// TIA Portal project "ACC_CONVEYOR" (V15)

(* hardware
DEVICE "ACC_CONVEYOR"  TP700 Comfort
   slot 0: "ACC_CONVEYOR"  TP700 Comfort  6AV2 124-0GC01-0AX0  14.0.0.0
   slot 1: "HMI_RT_1"  TP700 Comfort  6AV2 124-0GC01-0AX0  14.0.0.0
   slot 5: "ACC_CONVEYOR.IE_CP_1"  PROFINET Interface  14.0.0.0
      slot 1: "PROFINET Interface_1"  PROFINET Interface
         slot 1: "Port_1"  Port
         slot 2: "Port_2"  Port
   slot 7: "ACC_CONVEYOR.MPI/DP_CP_1"  MPI/DP Interface  14.0.0.0
*)

(* ===== HMI "HMI_RT_1" =====
system functions are stored by id; their names below are inferred from use
connection "SPS_1": IF1 B, SIMATIC S7 300/400 MPI

HMI tags "Default tag table"
   "bottleTypeNow" : Int AT %DB70.DBW10, 1 s
   "handmode_Key" : Byte AT %DB70.DBB38, 1 s
   "handMotorstat" : Int AT %DB70.DBW80, 1 s
   "keyGrup_a" : Byte AT %DB70.DBB0, 1 s
   "bottleTypeSelection" : Int AT %DB70.DBW170, 1 s
   "bottleAccSelect" : Bool AT %DB70.DBX2.5, 1 s
   "activeStart" : Bool AT %M10.0, 1 s
   "lubriState" : Bool AT %M48.0, 1 s
   "lubriCycle" : Int AT %DB51.DBW0, 1 s
   "lubriCycleinSec" : Int AT %DB51.DBW2, 1 s
   "lubriClockOP" : Bool AT %DB70.DBX8.0, 1 s
   "Contrass" : Int, internal

HMI tags "hardware_par"
   "select_motor" : Int AT %DB70.DBW40, 1 s
   "action" : Byte AT %DB70.DBB50, 1 s
   "copy" : Bool AT %DB70.DBX54.0, 1 s
   "towardsMotor" : Int AT %DB70.DBW52, 1 s
   "changeValue" : Int AT %DB70.DBW56, 1 s
   "value" : Real AT %DB70.DBD46, 1 s
   "parameter" : Int AT %DB70.DBW42, 1 s

HMI tags "software_par"
   "param_select" : Int AT %DB70.DBW30, 1 s
   "plc_Input" : Int AT %DB0.DBW30, 1 s
   "plc_Calc" : Int AT %DB0.DBW32, 1 s
   "plc_+fact" : Int AT %DB0.DBW34, 1 s
   "minim_Speed" : Int AT %DB0.DBW20, 1 s
   "maxim_Speed" : Int AT %DB0.DBW22, 1 s
   "corrLL" : Int AT %DB0.DBW8, 1 s
   "corrL" : Int AT %DB0.DBW10, 1 s
   "corrH" : Int AT %DB0.DBW12, 1 s
   "corrHH" : Int AT %DB0.DBW14, 1 s
   "frequency" : Int AT %DB0.DBW40, 1 s
   "rampUpSoft" : Int AT %DB0.DBW16, 1 s
   "rampDownSoft" : Int AT %DB0.DBW18, 1 s
   "fillUpLow" : Int AT %DB0.DBW0, 1 s
   "fillUpNomi" : Int AT %DB0.DBW2, 1 s
   "fillUpHigh" : Int AT %DB0.DBW4, 1 s
   "fillUpMaxi" : Int AT %DB0.DBW6, 1 s
   "statusDataWords" : Int AT %DB0.DBW0, 1 s
   "dbNumber" : Int AT %DB70.DBW180, 1 s
   "dwNumber" : Int AT %DB70.DBW182, 1 s
   "reff_Speed" : Int AT %DB0.DBW28, 1 s

HMI tags "regulation_EBI"
   "speedFiller" : Int AT %DB70.DBW90, 1 s
   "speedEBI" : Int AT %DB70.DBW92, 1 s
   "limOverNomin" : Int AT %DB0.DBW232, 1 s
   "limUnderNomin" : Int AT %DB0.DBW234, 1 s
   "correctionFact" : Int AT %DB0.DBW226, 1 s
   "maxSpeedEBI" : Int AT %DB0.DBW224, 1 s
   "minSpeedEBI" : Int AT %DB0.DBW230, 1 s
   "baseSpeed" : Int AT %DB0.DBW238, 1 s
   "btn_speedchange" : Byte AT %MB143, 1 s

HMI tags "inliner"
   "keyInlinerMode" : Byte AT %DB0.DBB278, 1 s
   "speedfilleer" : Int AT %DB0.DBW272, 1 s
   "speedInliner" : Int AT %DB0.DBW274, 1 s
   "limPosCorr" : Int AT %DB0.DBW246, 1 s
   "limNegCorr" : Int AT %DB0.DBW244, 1 s
   "stepPosCorr" : Int AT %DB0.DBW250, 1 s
   "stepNegCorr" : Int AT %DB0.DBW248, 1 s
   "missBotleRef" : Int AT %DB0.DBW240, 1 s
   "missBottleAct" : Int AT %DB0.DBW242, 1 s
   "actinlinerCorr" : Int AT %DB0.DBW266, 1 s
   "factFeeding" : Int AT %DB0.DBW10, 1 s
   "factInlliner" : Int AT %DB0.DBW12, 1 s
   "factOutfeed" : Int AT %DB0.DBW14, 1 s
   "fillUpFast" : Int AT %DB0.DBW254, 1 s
   "fillUpSlow" : Int AT %DB0.DBW252, 1 s
   "syncCorrStep" : Int AT %DB0.DBW280, 1 s
   "syncAfterBot" : Int AT %DB0.DBW282, 1 s
   "syncCounter" : Int AT %DB0.DBW284, 1 s
   "syncActCorr" : Int AT %DB0.DBW286, 1 s
   "syncStepNr" : Int AT %DB0.DBW288, 1 s

HMI tags "statistic"
   "totalMeasureTime" : DInt AT %DB70.DBD210, 1 s
   "lackBottlesInfeedFiller" : DInt AT %DB70.DBD214, 1 s
   "fillerStop" : DInt AT %DB70.DBD218, 1 s
   "fillerRunningBottleStopClosed" : DInt AT %DB70.DBD222, 1 s
   "startCounting" : Bool AT %DB70.DBX209.2, 1 s
   "stopCounting" : Bool AT %DB70.DBX209.3, 1 s
   "totalBottlesIntoFiller" : DInt AT %DB70.DBD226, 1 s
   "resetCounter" : Bool AT %DB70.DBX209.0, 1 s
   "confirm" : Bool AT %DB70.DBX209.1, 1 s
   "resetCounterState" : Bool AT %DB70.DBX208.0, 1 s

HMI tags "alarm"
   "alarm_1" : Int AT %DB70.DBW126, 1 s
   "alarm_2" : Int AT %DB70.DBW128, 1 s
   "alarm_3" : Int AT %DB70.DBW130, 1 s

HMI tags "monitor"
   "state_mot101" : Int AT %DB1.DBW56, 1 s
   "state_mot102" : Int AT %DB2.DBW56, 1 s
   "state_mot103" : Int AT %DB3.DBW56, 1 s
   "state_mot104" : Int AT %DB4.DBW56, 1 s
   "state_mot105" : Int AT %DB5.DBW56, 1 s
   "state_mot106" : Int AT %DB6.DBW56, 1 s
   "state_mot107" : Int AT %DB7.DBW56, 1 s
   "state_mot108" : Int AT %DB8.DBW56, 1 s
   "state_mot109" : Int AT %DB9.DBW56, 1 s
   "emc_1" : Bool AT %DB70.DBX168.0, 1 s
   "emc_2" : Bool AT %DB70.DBX168.1, 1 s
   "emc_3" : Bool AT %DB70.DBX168.2, 1 s
   "emc_4" : Bool AT %DB70.DBX168.3, 1 s
   "ebi_state" : Int AT %DB70.DBW200, 1 s
   "filler_state" : Int AT %DB70.DBW202, 1 s

discrete alarms
   2: 'MANUAL CONTROL ACTIVATED', class Status, trigger "alarm_1" bit 1
   3: 'LINE RUNNING', class Status, trigger "alarm_1" bit 2
   4: 'INLINER RECEPTABLE FULL', class Warnings, trigger "alarm_1" bit 3
   5: 'EMERGENCY STOP AT PANEL', class Errors, trigger "alarm_1" bit 4
      on Coming: ActivateScreen("121_DISPLAY_STATUS", 0)
   6: 'EMERGENCY STOP AT OUTFEED EBI', class Errors, trigger "alarm_1" bit 5
      on Coming: ActivateScreen("121_DISPLAY_STATUS", 0)
   7: 'EMERGENCY STOP AT INFEED FILLER', class Errors, trigger "alarm_1" bit 6
      on Coming: ActivateScreen("121_DISPLAY_STATUS", 0)
   8: 'FAULT ON MOTOR', class Errors, trigger "alarm_1" bit 7
      on Coming: ActivateScreen("121_DISPLAY_STATUS", 0)
   11: 'ACCUMULATION OUTFEED EBI', class Status, trigger "alarm_1" bit 10
   12: 'EBI NOT READY TO RUN', class Errors, trigger "alarm_1" bit 11
   13: 'EBI BOTTLESTOP MANUALLY OPENED', class Status, trigger "alarm_1" bit 12
   14: 'EBI AT MAXIMUM SPEED', class Warnings, trigger "alarm_1" bit 13
   15: 'EBI AT SYNCHRONISED SPEED', class Status, trigger "alarm_1" bit 14
   16: 'EBI AT MINIMUM SPEED', class Warnings, trigger "alarm_1" bit 15
   21: 'ACCUMULATION OUTFEED FILLER', class Status, trigger "alarm_2" bit 4
   22: 'FILLER STOP', class Errors, trigger "alarm_2" bit 5
   23: 'WAIT FOR FILLER TO OPEN BOTTLESTOP', class Status, trigger "alarm_2" bit 6
   31: 'INLINER RECEPTABLE ALMOT FULL', class Warnings, trigger "alarm_2" bit 14
   32: 'INLINER STOPPED RECEPTABLE FULL', class Warnings, trigger "alarm_2" bit 15
   33: 'INLINER FILLING UP', class Warnings, trigger "alarm_3" bit 0
   34: 'INLINER SYNCHRONISING', class Warnings, trigger "alarm_3" bit 1
   35: 'INLINER WAITS FOR BOTTLES', class Warnings, trigger "alarm_3" bit 2
   41: '..', class Warnings, trigger "alarm_3" bit 8

text list "motor_selection": 1 'motor 101'; 2 'motor 102'; 3 'motor 103'; 4 'motor 104'; 5 'motor 105'; 6 'motor 106'; 7 'motor 107'; 8 'motor 108'; 9 'motor 109'

text list "upload_download": 7 'Upload database to drive'; 6 'Download database from drive'

text list "hand_manual": 0 'MANUAL OFF'; 1 'MANUAL ON'

text list "bottle_type": 101 '620ml bottle'

text list "parameter": 1 'Motor power'; 2 'Motor voltage'; 3 'Motor frequency'; 4 'Motor current'; 5 'Min. frequency'; 6 'Max. frequency'; 7 'Ramp Up time'; 8 'Ramp Down time'; 9 'DP Address'; 10 'Actual frequency'; 11 'Actual current'; 12 'Actual'; 13 'Actual power KW'; 14 'Actual motor voltage'; 15 'Actual motor temperature'; 16 'Actual VLT temperature'; 17 'Actual Heat dispenser time'; 18 'Hours powered'; 19 'Hours running'; 20 'KWH counter'; 21 'latest fault code'

text list "valueParam": 1 'KW'; 2 'Volt'; 3 'HZ'; 4 'Amp'; 5 'HZ'; 6 'HZ'; 7 'sec.'; 8 'sec.'; 9 ''; 10 'HZ'; 11 'Amp'; 12 '%'; 13 'KW'; 14 'Volt'; 15 'Graden'; 16 'Graden'; 17 'Graden'; 18 'Uur'; 19 'Uur'; 20 'KWH'; 21 ''

Template "style_1" 800x480
   AlarmView "Template_Alarm view_1" at 0,0 size 800x27

screen "100_LOGO" 800x480, template "style_1"
   TextField "Text field_1" at 155,178 size 498x91; Text 'P A C K l N G'
   TextField "Text field_2" at 381,278 size 326x32; Text 'C R E A T I V E S Y S T E M S'
   Button "Button_1" at 3,28 size 792x446; TextOff '107_Trends'
      on Click: ActivateScreen("107_TRENDS_A", 0)

screen "104_HAND" 800x480, template "style_1"
   Button "btn_manualOFF" at 65,305 size 112x80; TextOff 'STOP MANUAL'; TextList "hand_manual"
      Appearance <- "handmode_Key"
      ProcessValue <- "handmode_Key"
      on Click: function_c82f6f27("handmode_Key", 0)
   Button "Button_3" at 200,414 size 99x66; TextOff 'Hardware Param'; Authorization "User administration"
      on Click: ActivateScreen("105_HARDWARE_PAR_1", 0)
   Button "Button_4" at 300,414 size 99x66; TextOff 'DW Status'; Authorization "User administration"
      on Click: ActivateScreen("122_DW_STATUS", 0)
   Button "Button_5" at 400,414 size 99x66; TextOff 'V_EBI Setup'; Authorization "User administration"
      on Click: ActivateScreen("118_V_EBI_SETUP", 0)
   Button "Button_6" at 500,414 size 99x66; TextOff 'Inline Setup'; Authorization "User administration"
      on Click: ActivateScreen("108_INLINER_1", 0)
   Button "Button_7" at 600,414 size 99x66; TextOff 'Software Param'; Authorization "User administration"
      on Click: ActivateScreen("119_SOFTWARE_PAR_1", 0)
   Button "Button_8" at 701,414 size 99x66; TextOff 'Main'
      on Click: ActivateScreen("107_TRENDS_A", 0)
   Button "btn_StartMan" at 648,59 size 112x80; TextOff 'START MANUAL'
      on Press: function_b14e0dd5("handmode_Key", 1)
   Button "btn_StopMan" at 648,154 size 112x80; TextOff 'STOP MANUAL'
      on Press: function_b14e0dd5("handmode_Key", 2)
   Button "btn_JOG" at 648,249 size 112x80; TextOff 'JOG'
      on Press: function_b14e0dd5("handmode_Key", 3)
   TextField "Text field_1" at 65,62 size 144x27; Text 'Manual Control :'
   TextField "Text field_2" at 65,123 size 58x27; Text 'Speed'
   TextField "Text field_3" at 26,163 size 36x27; Text 'akt.'
   TextField "Text field_4" at 24,203 size 40x27; Text 'reff.'
   IOField "actual_freq_motor" at 85,160 size 73x33; FormatPattern 99999
      ProcessValue <- "frequency"
   IOField "reff_speed_motor" at 85,200 size 73x33; FormatPattern 99999
      ProcessValue <- "reff_Speed"
   Bar "actual_frequency" at 219,148 size 340x64; MinimumValue 0; MaximumValue 100
      ProcessValue <- "frequency"
   SymbolicIOField "selection_motor" at 261,59 size 256x32; TextOff '0'; TextOn '1'; TextList "motor_selection"
      ProcessValue <- "param_select"
   TextField "Text field_5" at 167,163 size 58x27; Text 'Speed / HZ'
   Circle "motor_101" at 250,248 size 29x29
      Appearance <- "handMotorstat"
   Circle "motor_102" at 282,248 size 29x29
      Appearance <- "handMotorstat"
   Circle "motor_103" at 314,248 size 29x29
      Appearance <- "handMotorstat"
   Circle "motor_104" at 346,248 size 29x29
      Appearance <- "handMotorstat"
   Circle "motor_105" at 378,248 size 29x29
      Appearance <- "handMotorstat"
   Circle "motor_106" at 410,248 size 29x29
      Appearance <- "handMotorstat"
   Circle "motor_107" at 442,248 size 29x29
      Appearance <- "handMotorstat"
   Circle "motor_108" at 474,248 size 29x29
      Appearance <- "handMotorstat"
   Circle "motor_109" at 506,248 size 29x29
      Appearance <- "handMotorstat"
   TextField "Text field_8" at 255,277 size 19x23; Text 'reff. / 1'
   TextField "Text field_9" at 287,277 size 19x23; Text 'reff. / 2'
   TextField "Text field_10" at 319,277 size 19x23; Text 'reff. / 3'
   TextField "Text field_11" at 351,277 size 19x23; Text 'reff. / 4'
   TextField "Text field_12" at 383,277 size 19x23; Text 'reff. / 5'
   TextField "Text field_13" at 415,277 size 19x23; Text 'reff. / 6'
   TextField "Text field_14" at 447,277 size 19x23; Text 'reff. / 7'
   TextField "Text field_15" at 479,277 size 19x23; Text 'reff. / 8'
   TextField "Text field_16" at 511,277 size 19x23; Text 'reff. / 9'
   TextField "Text field_17" at 216,253 size 28x23; Text 'reff. / 60'
   Button "Button_1" at 0,414 size 99x66; TextOff 'Start'
      on Press: function_b14e0dd5("keyGrup_a", 0)
      Appearance <- "activeStart"
   Button "Button_2" at 100,414 size 99x66; TextOff 'Stop'
      on Press: function_b14e0dd5("keyGrup_a", 1)

screen "105_HARDWARE_PAR_1" 800x480, template "style_1"
   Button "Button_6" at 500,414 size 99x66; TextOff 'Param 2'
      on Click: ActivateScreen("110_HARDWARE_PAR_2", 0)
   TextField "Text field_1" at 100,46 size 139x27; Text 'Read or modify'
   TextField "Text field_2" at 100,94 size 97x27; Text 'Parameter'
   TextField "Text field_3" at 100,143 size 57x27; Text 'Value'
   Button "Button_9" at 100,272 size 136x53; TextOff 'Stop / Read out'
      on Press: function_b14e0dd5("action", 2)
   Button "Button_10" at 100,337 size 136x53; TextOff 'Stop / Modify'
      on Press: function_b14e0dd5("action", 3)
   Button "Button_11" at 328,272 size 136x53; TextOff 'Stop / +'
      on Press: function_b14e0dd5("action", 0)
   Button "Button_12" at 328,337 size 136x53; TextOff 'Stop / -'
      on Press: function_b14e0dd5("action", 1)
   Button "Button_13" at 556,272 size 143x53; TextOff 'Stop / Save in DB'
      on Click: function_b3f726e6("action", 4)
   Button "Button_14" at 556,337 size 142x53; TextOff 'Stop / Read from DB'
      on Click: function_b3f726e6("action", 5)
   IOField "I/O field_1" at 328,140 size 107x33; FormatPattern 9999.99
      ProcessValue <- "value"
   SymbolicIOField "Symbolic I/O field_3" at 450,140 size 170x32; TextOn '1'; TextOff '0'; TextList "valueParam"
      ProcessValue <- "parameter"
   SymbolicIOField "Symbolic I/O field_1" at 328,43 size 259x32; TextOn '1'; TextOff '0'; TextList "motor_selection"
      ProcessValue <- "select_motor"
   Button "Button_4" at 300,414 size 99x66; TextOff 'DW Status K4'
      on Press: function_b14e0dd5("keyGrup_a", 3)
   Button "Button_5" at 400,414 size 99x66; TextOff 'V_EBI Setup K5'
      on Press: function_b14e0dd5("keyGrup_a", 4)
   Button "Button_8" at 701,414 size 99x66; TextOff 'Main'
      on Click: ActivateScreen("107_TRENDS_A", 0)
   Button "Button_1" at 0,414 size 99x66; TextOff 'Start'
      on Press: function_b14e0dd5("keyGrup_a", 0)
      Appearance <- "activeStart"
   Button "Button_2" at 100,414 size 99x66; TextOff 'Stop'
      on Press: function_b14e0dd5("keyGrup_a", 1)
   Button "Button_3" at 200,414 size 99x66; TextOff 'Stop / K3'
      on Press: function_b14e0dd5("keyGrup_a", 2)
   Button "Button_7" at 600,414 size 99x66; TextOff 'Software Param K7'
      on Press: function_b14e0dd5("keyGrup_a", 6)
   Button "Button_15" at 277,202 size 70x34; TextOff 'DW Status'
      on Click: function_dd21b452("changeValue", 1)
   Button "Button_16" at 427,202 size 70x34; TextOff 'DW Status'
      on Click: function_b9b71300("changeValue", 1)
   SymbolicIOField "Symbolic I/O field_2" at 328,91 size 371x32; TextOn '1'; TextOff '0'; TextList "parameter"
      ProcessValue <- "parameter"
   GraphicView "Graphic view_1" at 393,197 size 34x39; Picture "panah'"
      HorizontalMovement <- "changeValue"

screen "113_UTILITY" 800x480, template "style_1"
   Button "Button_1" at 0,414 size 99x66; TextOff 'Start'
      on Press: function_b14e0dd5("keyGrup_a", 0)
      Appearance <- "activeStart"
   Button "Button_2" at 100,414 size 99x66; TextOff 'Stop'
      on Press: function_b14e0dd5("keyGrup_a", 1)
   Button "Button_3" at 200,414 size 149x66; TextOff 'Hardware Param Contras -'
      on Click: function_b9b71300("Contrass", 1)
      on Change: function_e4c2bb66("Contrass")
   Button "Button_4" at 351,414 size 148x66; TextOff 'DW Status Contras +'
      on Click: function_dd21b452("Contrass", 1)
      on Change: function_e4c2bb66("Contrass")
   Button "Button_6" at 500,414 size 99x66; TextOff 'Clean Screen'
      on Click: function_be740847(30)
   Button "Button_7" at 600,414 size 99x66; TextOff 'Software Param Calibrate Screen'
      on Click: function_bc3e350c()
   Button "Button_8" at 701,414 size 99x66; TextOff 'Main'
      on Click: ActivateScreen("107_TRENDS_A", 0)
   Button "Button_5" at 118,291 size 154x63; TextOff 'Software Param Status'
      on Click: ActivateScreen("121_DISPLAY_STATUS", 0)
   Button "Button_9" at 526,290 size 154x63; TextOff 'Software Param Statistics'
      on Click: ActivateScreen("117_STATISTICS", 0)
   TextField "Text field_2" at 98,152 size 107x27; Text 'Speed / Lubrification'
   TextField "Text field_1" at 275,193 size 58x27; Text 'Speed / Cycle'
   TextField "Text field_3" at 448,193 size 103x27; Text 'Speed / Sec.in cycle'
   Circle "Circle_1" at 382,152 size 29x29
      Appearance <- "lubriState"
   IOField "I/O field_1" at 271,150 size 73x33; FormatPattern 9999
      ProcessValue <- "lubriCycle"
   IOField "I/O field_2" at 450,150 size 73x33; FormatPattern 9999
      ProcessValue <- "lubriCycleinSec"
   TextField "Text field_4" at 177,61 size 58x27; Text 'Speed / Clock'
   Button "Button_10" at 537,43 size 154x59; TextOff 'Software Param Clock OP --> PLC'
      on Press: function_b14e0dd5("lubriClockOP", 0)
   DateTimeField "Date/time field_1" at 284,58 size 215x32

screen "117_STATISTICS" 800x480, template "style_1"
   Button "btn_resetcounter" at 297,414 size 202x66; TextOff 'DW Status RESET COUNTER'
      on Press: function_b14e0dd5("resetCounter", 0)
      Appearance <- "resetCounterState"
   Button "btn_confirm" at 499,414 size 202x66; TextOff 'CONFIRM'
      on Press: function_b14e0dd5("confirm", 0)
   Button "Button_8" at 701,414 size 99x66; TextOff 'Main'
      on Click: ActivateScreen("107_TRENDS_A", 0)
   TextField "Text field_2" at 267,62 size 191x27; Text 'Speed / Total measure time :'
   TextField "Text field_1" at 217,103 size 241x27; Text 'Speed / Lack of bottle infeed filler :'
   TextField "Text field_3" at 313,144 size 145x27; Text 'Speed / Filler Stopped :'
   TextField "Text field_4" at 165,185 size 293x27; Text 'Speed / Filler running, bottlestop closed :'
   TextField "Text field_5" at 248,348 size 210x27; Text 'Speed / Total bottles into filler :'
   Button "btn_stopcounting" at 373,241 size 150x66; TextOff 'Stop Stop Counting'
      on Press: function_b14e0dd5("stopCounting", 0)
   Button "btn_startcounting" at 214,241 size 150x66; TextOff 'Start Start Counting'
      on Press: function_b14e0dd5("startCounting", 0)
   IOField "I/O field_1" at 466,59 size 93x33; FormatPattern 9999999
      ProcessValue <- "totalMeasureTime"
   IOField "I/O field_2" at 466,100 size 93x33; FormatPattern 9999999
      ProcessValue <- "lackBottlesInfeedFiller"
   IOField "I/O field_3" at 466,141 size 93x33; FormatPattern 9999999
      ProcessValue <- "fillerStop"
   IOField "I/O field_4" at 466,182 size 93x33; FormatPattern 9999999
      ProcessValue <- "fillerRunningBottleStopClosed"
   IOField "I/O field_5" at 466,345 size 93x33; FormatPattern 9999999
      ProcessValue <- "totalBottlesIntoFiller"
   TextField "Text field_6" at 572,62 size 34x27; Text 'Speed / Sec'
   TextField "Text field_7" at 572,103 size 34x27; Text 'Speed / Sec'
   TextField "Text field_8" at 572,144 size 34x27; Text 'Speed / Sec'
   TextField "Text field_9" at 572,185 size 34x27; Text 'Speed / Sec'
   Button "Button_1" at 0,414 size 99x66; TextOff 'Start'
      on Press: function_b14e0dd5("keyGrup_a", 0)
      Appearance <- "activeStart"
   Button "Button_2" at 99,414 size 99x66; TextOff 'Stop'
      on Press: function_b14e0dd5("keyGrup_a", 1)
   Button "Button_3" at 198,414 size 99x66; TextOff 'Stop / K3'
      on Press: function_b14e0dd5("keyGrup_a", 2)

screen "108_INLINER_1" 800x480, template "style_1"
   Bar "missbottleact" at 604,96 size 39x265; MinimumValue 0; MaximumValue 10
      ProcessValue <- "missBottleAct"
   Button "btn_Sync2" at 330,149 size 99x66; TextOff 'Hardware Param Sync'
      on Click: function_c82f6f27("keyInlinerMode", 3)
      Visibility <- "keyInlinerMode"
   Button "btn_fillUptact2" at 330,221 size 99x66; TextOff 'Hardware Param Fill up tact'
      on Click: function_c82f6f27("keyInlinerMode", 4)
      Visibility <- "keyInlinerMode"
   Button "btn_fillUptime2" at 330,293 size 99x66; TextOff 'Hardware Param Fill up time'
      on Click: function_c82f6f27("keyInlinerMode", 5)
      Visibility <- "keyInlinerMode"
   Button "btn_autoReset2" at 330,77 size 99x66; TextOff 'Hardware Param Auto Reset'
      on Click: function_c82f6f27("keyInlinerMode", 2)
      Visibility <- "keyInlinerMode"
   TextField "Text field_2" at 21,36 size 173x27; Text 'Speed / Inliner Setup/Status'
   TextField "Text field_1" at 21,85 size 112x27; Text 'Speed / Speed filler :'
   TextField "Text field_3" at 21,116 size 128x27; Text 'Speed / Speed inliner :'
   TextField "Text field_4" at 21,147 size 121x27; Text 'Speed / Lim.pos.corr :'
   TextField "Text field_5" at 21,178 size 124x27; Text 'Speed / Lim.neg.corr :'
   TextField "Text field_6" at 21,209 size 130x27; Text 'Speed / Step.pos.corr :'
   TextField "Text field_7" at 21,240 size 133x27; Text 'Speed / Step.neg.corr :'
   TextField "Text field_8" at 21,271 size 153x27; Text 'Speed / Miss. bottle reff. :'
   TextField "Text field_9" at 21,302 size 149x27; Text 'Speed / Miss. bottle act. :'
   Button "Button_4" at 300,414 size 99x66; TextOff 'DW Status'; Authorization "User administration"
      on Click: ActivateScreen("122_DW_STATUS", 0)
   Button "Button_5" at 400,414 size 99x66; TextOff 'V_EBI Setup V_EBI setup'; Authorization "User administration"
      on Click: ActivateScreen("118_V_EBI_SETUP", 0)
   Button "Button_6" at 500,414 size 99x66; TextOff 'Software Param'; Authorization "User administration"
      on Click: ActivateScreen("119_SOFTWARE_PAR_1", 0)
   Button "Button_7" at 600,414 size 99x66; TextOff 'Software Param Inline page 2'; Authorization "User administration"
      on Click: ActivateScreen("109_INLINER_2", 0)
   Button "Button_8" at 701,414 size 99x66; TextOff 'Main'
      on Click: ActivateScreen("107_TRENDS_A", 0)
   Button "btn_autoReset" at 330,77 size 99x66; TextOff 'Hardware Param Auto Reset'
      on Click: function_c82f6f27("keyInlinerMode", 2)
      Visibility <- "keyInlinerMode"
   Button "btn_Sync" at 330,149 size 99x66; TextOff 'Hardware Param Sync'
      on Click: function_c82f6f27("keyInlinerMode", 3)
      Visibility <- "keyInlinerMode"
   Button "btn_fillUptact" at 330,221 size 99x66; TextOff 'Hardware Param Fill up tact'
      on Click: function_c82f6f27("keyInlinerMode", 4)
      Visibility <- "keyInlinerMode"
   Button "btn_fillUptime" at 330,293 size 99x66; TextOff 'Hardware Param Fill up time'
      on Click: function_c82f6f27("keyInlinerMode", 5)
      Visibility <- "keyInlinerMode"
   IOField "I/O field_1" at 212,82 size 73x33; FormatPattern 99999
      ProcessValue <- "speedfilleer"
   IOField "I/O field_2" at 212,113 size 73x33; FormatPattern 99999
      ProcessValue <- "speedInliner"
   IOField "I/O field_3" at 212,144 size 73x33; FormatPattern 99999
      ProcessValue <- "limPosCorr"
   IOField "I/O field_4" at 212,175 size 73x33; FormatPattern 99999
      ProcessValue <- "limNegCorr"
   IOField "I/O field_5" at 212,206 size 73x33; FormatPattern 99999
      ProcessValue <- "stepPosCorr"
   IOField "I/O field_6" at 212,237 size 73x33; FormatPattern 99999
      ProcessValue <- "stepNegCorr"
   IOField "I/O field_7" at 212,268 size 73x33; FormatPattern 99999
      ProcessValue <- "missBotleRef"
   IOField "I/O field_8" at 548,37 size 53x33; FormatPattern 99999
      ProcessValue <- "missBotleRef"
   IOField "I/O field_9" at 600,37 size 53x33; FormatPattern 99999
      ProcessValue <- "missBottleAct"
   IOField "I/O field_10" at 652,37 size 53x33; FormatPattern 99999
      ProcessValue <- "actinlinerCorr"
   Bar "missbottlereff" at 542,84 size 73x289; MinimumValue 0; MaximumValue 10
      ProcessValue <- "missBotleRef"
   Bar "correction" at 643,84 size 89x289; MinimumValue -99; MaximumValue 180
      MaximumValue <- "limPosCorr"
      MinimumValue <- "limNegCorr"
      ProcessValue <- "actinlinerCorr"
   TextField "Text field_13" at 364,37 size 177x33; Text 'Speed / 620ml bottle'
   IOField "I/O field_11" at 212,299 size 73x33; FormatPattern 99999
      ProcessValue <- "missBottleAct"
   Button "Button_1" at 0,414 size 99x66; TextOff 'Start'
      on Press: function_b14e0dd5("keyGrup_a", 0)
      Appearance <- "activeStart"
   Button "Button_2" at 100,414 size 99x66; TextOff 'Stop'
      on Press: function_b14e0dd5("keyGrup_a", 1)
   Button "Button_3" at 200,414 size 99x66; TextOff 'Stop / K3'
      on Press: function_b14e0dd5("keyGrup_a", 2)
   TextField "Text field_10" at 541,375 size 58x27; Text 'Speed / Reff.'
   TextField "Text field_11" at 595,375 size 58x27; Text 'Speed / Act.'
   TextField "Text field_12" at 664,375 size 58x27; Text 'Speed / Corr.'

screen "112_INLINER_3" 800x480, template "style_1"
   TextField "Text field_4" at 21,147 size 144x27; Text 'Speed / Sync.corr. step :'
   TextField "Text field_5" at 21,179 size 136x27; Text 'Speed / Sync.after bot :'
   TextField "Text field_6" at 21,211 size 128x27; Text 'Speed / Sync.counter :'
   TextField "Text field_7" at 21,243 size 139x27; Text 'Speed / Sync.actu.corr :'
   TextField "Text field_8" at 21,275 size 123x27; Text 'Speed / Sync.step.nr :'
   TextField "Text field_2" at 21,36 size 173x27; Text 'Speed / Inliner Setup/Status'
   TextField "Text field_1" at 21,85 size 112x27; Text 'Speed / Speed filler :'
   TextField "Text field_3" at 21,116 size 128x27; Text 'Speed / Speed inliner :'
   Button "Button_7" at 600,414 size 99x66; TextOff 'Software Param Inliner page 1'; Authorization "User administration"
      on Click: ActivateScreen("108_INLINER_1", 0)
   Button "Button_8" at 701,414 size 99x66; TextOff 'Main'
      on Click: ActivateScreen("107_TRENDS_A", 0)
   IOField "I/O field_1" at 212,82 size 73x33; FormatPattern 99999
      ProcessValue <- "speedfilleer"
   IOField "I/O field_2" at 212,113 size 73x33; FormatPattern 99999
      ProcessValue <- "speedInliner"
   IOField "I/O field_3" at 212,144 size 73x33; FormatPattern 99999
      ProcessValue <- "syncCorrStep"
   IOField "I/O field_4" at 212,175 size 73x33; FormatPattern 99999
      ProcessValue <- "syncAfterBot"
   IOField "I/O field_5" at 212,206 size 73x33; FormatPattern 99999
      ProcessValue <- "syncCounter"
   IOField "I/O field_6" at 212,237 size 73x33; FormatPattern 99999
      ProcessValue <- "syncActCorr"
   IOField "I/O field_7" at 212,268 size 73x33; FormatPattern 99999
      ProcessValue <- "syncStepNr"
   TextField "Text field_13" at 364,37 size 177x33; Text 'Speed / 620ml bottle'
   Button "Button_4" at 300,414 size 99x66; TextOff 'DW Status'; Authorization "User administration"
      on Click: ActivateScreen("122_DW_STATUS", 0)
   Button "Button_5" at 400,414 size 99x66; TextOff 'V_EBI Setup V_EBI setup'; Authorization "User administration"
      on Click: ActivateScreen("118_V_EBI_SETUP", 0)
   Button "Button_6" at 500,414 size 99x66; TextOff 'Software Param'; Authorization "User administration"
      on Click: ActivateScreen("119_SOFTWARE_PAR_1", 0)
   IOField "I/O field_8" at 548,37 size 53x33; FormatPattern 99999
      ProcessValue <- "missBotleRef"
   IOField "I/O field_9" at 600,37 size 53x33; FormatPattern 99999
      ProcessValue <- "missBottleAct"
   IOField "I/O field_10" at 652,37 size 53x33; FormatPattern 99999
      ProcessValue <- "actinlinerCorr"
   TextField "Text field_10" at 541,375 size 58x27; Text 'Speed / Reff.'
   TextField "Text field_11" at 595,375 size 58x27; Text 'Speed / Act.'
   TextField "Text field_12" at 664,375 size 58x27; Text 'Speed / Corr.'
   Button "Button_1" at 0,414 size 99x66; TextOff 'Start'
      on Press: function_b14e0dd5("keyGrup_a", 0)
      Appearance <- "activeStart"
   Button "Button_2" at 100,414 size 99x66; TextOff 'Stop'
      on Press: function_b14e0dd5("keyGrup_a", 1)
   Button "Button_3" at 200,414 size 99x66; TextOff 'Stop / K3'
      on Press: function_b14e0dd5("keyGrup_a", 2)
   Bar "Bar_2" at 604,96 size 39x265; MinimumValue 0; MaximumValue 10
      ProcessValue <- "missBottleAct"
   Button "Button_14" at 330,149 size 99x66; TextOff 'Hardware Param Sync'
      on Click: function_c82f6f27("keyInlinerMode", 3)
      Visibility <- "keyInlinerMode"
   Button "Button_15" at 330,221 size 99x66; TextOff 'Hardware Param Fill up tact'
      on Click: function_c82f6f27("keyInlinerMode", 4)
      Visibility <- "keyInlinerMode"
   Button "Button_16" at 330,293 size 99x66; TextOff 'Hardware Param Fill up time'
      on Click: function_c82f6f27("keyInlinerMode", 5)
      Visibility <- "keyInlinerMode"
   Button "Button_13" at 330,77 size 99x66; TextOff 'Hardware Param Auto Reset'
      on Click: function_c82f6f27("keyInlinerMode", 2)
      Visibility <- "keyInlinerMode"
   Button "Button_9" at 330,77 size 99x66; TextOff 'Hardware Param Auto Reset'
      on Click: function_c82f6f27("keyInlinerMode", 2)
      Visibility <- "keyInlinerMode"
   Button "Button_10" at 330,149 size 99x66; TextOff 'Hardware Param Sync'
      on Click: function_c82f6f27("keyInlinerMode", 3)
      Visibility <- "keyInlinerMode"
   Button "Button_11" at 330,221 size 99x66; TextOff 'Hardware Param Fill up tact'
      on Click: function_c82f6f27("keyInlinerMode", 4)
      Visibility <- "keyInlinerMode"
   Button "Button_12" at 330,292 size 99x66; TextOff 'Hardware Param Fill up time'
      on Click: function_c82f6f27("keyInlinerMode", 5)
      Visibility <- "keyInlinerMode"
   Bar "Bar_1" at 542,84 size 73x289; MinimumValue 0; MaximumValue 10
      ProcessValue <- "missBotleRef"
   Bar "Bar_3" at 643,84 size 89x289; MinimumValue -99; MaximumValue 180
      MinimumValue <- "limNegCorr"
      ProcessValue <- "actinlinerCorr"
      MaximumValue <- "limPosCorr"

screen "109_INLINER_2" 800x480, template "style_1"
   TextField "Text field_4" at 21,147 size 128x27; Text 'Speed / Fact. feeding :'
   TextField "Text field_5" at 21,178 size 116x27; Text 'Speed / Fact. inliner :'
   TextField "Text field_6" at 21,209 size 129x27; Text 'Speed / Fact. outfeed :'
   TextField "Text field_7" at 21,240 size 104x27; Text 'Speed / Fill up fast :'
   TextField "Text field_8" at 21,271 size 110x27; Text 'Speed / Fill up slow :'
   TextField "Text field_2" at 21,36 size 173x27; Text 'Speed / Inliner Setup/Status'
   TextField "Text field_1" at 21,85 size 112x27; Text 'Speed / Speed filler :'
   TextField "Text field_3" at 21,116 size 128x27; Text 'Speed / Speed inliner :'
   Button "Button_7" at 600,414 size 99x66; TextOff 'Software Param Inliner page 3'; Authorization "User administration"
      on Click: ActivateScreen("112_INLINER_3", 0)
   Button "Button_8" at 701,414 size 99x66; TextOff 'Main'
      on Click: ActivateScreen("107_TRENDS_A", 0)
   IOField "I/O field_1" at 212,82 size 73x33; FormatPattern 99999
      ProcessValue <- "speedfilleer"
   IOField "I/O field_2" at 212,113 size 73x33; FormatPattern 99999
      ProcessValue <- "speedInliner"
   IOField "I/O field_3" at 212,144 size 73x33; FormatPattern 99999
      ProcessValue <- "factFeeding"
   IOField "I/O field_4" at 212,175 size 73x33; FormatPattern 99999
      ProcessValue <- "factInlliner"
   IOField "I/O field_5" at 212,206 size 73x33; FormatPattern 99999
      ProcessValue <- "factOutfeed"
   IOField "I/O field_6" at 212,237 size 73x33; FormatPattern 99999
      ProcessValue <- "fillUpFast"
   IOField "I/O field_7" at 212,268 size 73x33; FormatPattern 99999
      ProcessValue <- "fillUpSlow"
   TextField "Text field_13" at 364,37 size 177x33; Text 'Speed / 620ml bottle'
   Button "Button_4" at 300,414 size 99x66; TextOff 'DW Status'; Authorization "User administration"
      on Click: ActivateScreen("122_DW_STATUS", 0)
   Button "Button_5" at 400,414 size 99x66; TextOff 'V_EBI Setup V_EBI setup'; Authorization "User administration"
      on Click: ActivateScreen("118_V_EBI_SETUP", 0)
   Button "Button_6" at 500,414 size 99x66; TextOff 'Software Param'; Authorization "User administration"
      on Click: ActivateScreen("119_SOFTWARE_PAR_1", 0)
   IOField "I/O field_8" at 548,37 size 53x33; FormatPattern 99999
      ProcessValue <- "missBotleRef"
   IOField "I/O field_9" at 600,37 size 53x33; FormatPattern 99999
      ProcessValue <- "missBottleAct"
   IOField "I/O field_10" at 652,37 size 53x33; FormatPattern 99999
      ProcessValue <- "actinlinerCorr"
   Button "Button_1" at 0,414 size 99x66; TextOff 'Start'
      on Press: function_b14e0dd5("keyGrup_a", 0)
      Appearance <- "activeStart"
   Button "Button_2" at 100,414 size 99x66; TextOff 'Stop'
      on Press: function_b14e0dd5("keyGrup_a", 1)
   Button "Button_3" at 200,414 size 99x66; TextOff 'Stop / K3'
      on Press: function_b14e0dd5("keyGrup_a", 2)
   TextField "Text field_10" at 541,375 size 58x27; Text 'Speed / Reff.'
   TextField "Text field_11" at 595,375 size 58x27; Text 'Speed / Act.'
   TextField "Text field_12" at 664,375 size 58x27; Text 'Speed / Corr.'
   Bar "Bar_2" at 604,96 size 39x265; MinimumValue 0; MaximumValue 10
      ProcessValue <- "missBottleAct"
   Button "Button_14" at 330,149 size 99x66; TextOff 'Hardware Param Sync'
      on Click: function_c82f6f27("keyInlinerMode", 3)
      Visibility <- "keyInlinerMode"
   Button "Button_15" at 330,221 size 99x66; TextOff 'Hardware Param Fill up tact'
      on Click: function_c82f6f27("keyInlinerMode", 4)
      Visibility <- "keyInlinerMode"
   Button "Button_16" at 330,293 size 99x66; TextOff 'Hardware Param Fill up time'
      on Click: function_c82f6f27("keyInlinerMode", 5)
      Visibility <- "keyInlinerMode"
   Button "Button_13" at 330,77 size 99x66; TextOff 'Hardware Param Auto Reset'
      on Click: function_c82f6f27("keyInlinerMode", 2)
      Visibility <- "keyInlinerMode"
   Button "Button_9" at 330,77 size 99x66; TextOff 'Hardware Param Auto Reset'
      on Click: function_c82f6f27("keyInlinerMode", 2)
      Visibility <- "keyInlinerMode"
   Button "Button_10" at 330,149 size 99x66; TextOff 'Hardware Param Sync'
      on Click: function_c82f6f27("keyInlinerMode", 3)
      Visibility <- "keyInlinerMode"
   Button "Button_11" at 330,221 size 99x66; TextOff 'Hardware Param Fill up tact'
      on Click: function_c82f6f27("keyInlinerMode", 4)
      Visibility <- "keyInlinerMode"
   Button "Button_12" at 330,293 size 99x66; TextOff 'Hardware Param Fill up time'
      on Click: function_c82f6f27("keyInlinerMode", 5)
      Visibility <- "keyInlinerMode"
   Bar "Bar_1" at 542,84 size 73x289; MinimumValue 0; MaximumValue 10
      ProcessValue <- "missBotleRef"
   Bar "Bar_3" at 643,84 size 89x289; MinimumValue -99; MaximumValue 180
      MinimumValue <- "limNegCorr"
      ProcessValue <- "actinlinerCorr"
      MaximumValue <- "limPosCorr"

screen "111_HARDWARE_PAR_3" 800x480, template "style_1"
   Button "Button_6" at 500,414 size 99x66; TextOff 'Param 1'
      on Click: ActivateScreen("105_HARDWARE_PAR_1", 0)
   Button "Button_7" at 600,414 size 99x66; TextOff 'Software Param Param 2'
      on Click: ActivateScreen("110_HARDWARE_PAR_2", 0)
   TextField "Text field_1" at 161,75 size 165x27; Text 'Copy values motor'
   TextField "Text field_2" at 161,188 size 126x27; Text 'towards motor'
   Button "Button_9" at 300,282 size 194x53; TextOff 'Stop / Copy'
      on Press: function_b14e0dd5("copy", 0)
   Button "Button_4" at 300,414 size 99x66; TextOff 'DW Status K4'
      on Press: function_b14e0dd5("keyGrup_a", 3)
   Button "Button_5" at 400,414 size 99x66; TextOff 'V_EBI Setup K5'
      on Press: function_b14e0dd5("keyGrup_a", 4)
   Button "Button_8" at 701,414 size 99x66; TextOff 'Main'
      on Click: ActivateScreen("107_TRENDS_A", 0)
   Button "Button_1" at 0,414 size 99x66; TextOff 'Start'
      on Press: function_b14e0dd5("keyGrup_a", 0)
      Appearance <- "activeStart"
   Button "Button_2" at 100,414 size 99x66; TextOff 'Stop'
      on Press: function_b14e0dd5("keyGrup_a", 1)
   Button "Button_3" at 200,414 size 99x66; TextOff 'Stop / K3'
      on Press: function_b14e0dd5("keyGrup_a", 2)
   SymbolicIOField "Symbolic I/O field_1" at 346,72 size 259x32; TextOn '1'; TextOff '0'; TextList "motor_selection"
      ProcessValue <- "select_motor"
   SymbolicIOField "Symbolic I/O field_2" at 346,185 size 259x32; TextOn '1'; TextOff '0'; TextList "motor_selection"
      ProcessValue <- "towardsMotor"

screen "110_HARDWARE_PAR_2" 800x480, template "style_1"
   Button "Button_6" at 500,414 size 99x66; TextOff 'Param 3'
      on Click: ActivateScreen("111_HARDWARE_PAR_3", 0)
   Button "Button_7" at 600,414 size 99x66; TextOff 'Software Param Param 1'
      on Click: ActivateScreen("105_HARDWARE_PAR_1", 0)
   TextField "Text field_1" at 136,75 size 121x27; Text 'Modify motor'
   TextField "Text field_2" at 201,178 size 56x27; Text 'Action'
   Button "Button_9" at 187,275 size 143x53; TextOff 'Stop / Download'
      on Press: function_b14e0dd5("action", 2)
   Button "Button_10" at 477,275 size 143x53; TextOff 'Stop / Upload'
      on Press: function_b14e0dd5("action", 3)
   SymbolicIOField "Symbolic I/O field_1" at 292,72 size 259x32; TextOn '1'; TextOff '0'; TextList "motor_selection"
      ProcessValue <- "select_motor"
   SymbolicIOField "Symbolic I/O field_2" at 292,175 size 323x32; TextOn '1'; TextOff '0'; TextList "upload_download"
      ProcessValue <- "action"
   Button "Button_4" at 300,414 size 99x66; TextOff 'DW Status K4'
      on Press: function_b14e0dd5("keyGrup_a", 3)
   Button "Button_5" at 400,414 size 99x66; TextOff 'V_EBI Setup K5'
      on Press: function_b14e0dd5("keyGrup_a", 4)
   Button "Button_8" at 701,414 size 99x66; TextOff 'Main'
      on Click: ActivateScreen("107_TRENDS_A", 0)
   Button "Button_1" at 0,414 size 99x66; TextOff 'Start'
      on Press: function_b14e0dd5("keyGrup_a", 0)
      Appearance <- "activeStart"
   Button "Button_2" at 100,414 size 99x66; TextOff 'Stop'
      on Press: function_b14e0dd5("keyGrup_a", 1)
   Button "Button_3" at 200,414 size 99x66; TextOff 'Stop / K3'
      on Press: function_b14e0dd5("keyGrup_a", 2)

screen "107_TRENDS_A" 800x480, template "style_1"
   Button "Button_3" at 200,414 size 99x66; TextOff 'Hardware Param Bottle type'
      on Click: ActivateScreen("106_BOTTLE_TYPE", 0)
   Button "Button_4" at 300,414 size 99x66; TextOff 'DW Status Utility'
      on Click: ActivateScreen("113_UTILITY", 0)
   Button "Button_5" at 400,414 size 99x66; TextOff 'V_EBI Setup Messages'
      on Click: ActivateScreen("116_MESSAGES", 0)
   Button "Button_6" at 500,414 size 99x66; TextOff 'Param'
      on Click: ActivateScreen("115_TRENDS_B", 0)
   Button "Button_7" at 600,414 size 99x66; TextOff 'Software Param Hand'; Authorization "User administration"
      on Click: ActivateScreen("104_HAND", 0)
   Button "Button_8" at 701,414 size 99x66; TextOff 'Main'
      on Click: ActivateScreen("100_LOGO", 0)
   TextField "Text field_1" at 18,381 size 58x27; Text 'Speed / Filler :'
   TextField "Text field_2" at 594,381 size 58x27; Text 'Speed / EBI :'
   TextField "Text field_3" at 123,379 size 70x32; Text 'Speed / 000 b/h'
   TextField "Text field_4" at 698,379 size 70x32; Text 'Speed / 000 b/h'
   TrendView "Trend view_1" at 9,67 size 785x283
   IOField "I/O field_1" at 74,379 size 47x32; FormatPattern 99999
      ProcessValue <- "speedFiller"
   IOField "I/O field_2" at 651,379 size 47x32; FormatPattern 99999
      ProcessValue <- "speedEBI"
   Button "Button_9" at 6,364 size 786x49; TextOff 'monitor'
      on Click: ActivateScreen("121_DISPLAY_STATUS", 0)
   TextField "Text field_12" at 22,30 size 166x33; Text 'Speed / 620ml bottle'
   Button "Button_1" at 0,414 size 99x66; TextOff 'Start'
      on Press: function_b14e0dd5("keyGrup_a", 0)
      Appearance <- "activeStart"
   Button "Button_2" at 100,414 size 99x66; TextOff 'Stop'
      on Press: function_b14e0dd5("keyGrup_a", 1)

screen "106_BOTTLE_TYPE" 800x480, template "style_1"
   TextField "Text field_1" at 21,43 size 134x27; Text 'Speed / Actual selection'
   TextField "Text field_2" at 201,204 size 113x27; Text 'Speed / Bottle type :'
   SymbolicIOField "bottletype_selection" at 333,202 size 247x32; TextOn '1'; TextOff '0'; TextList "bottle_type"
      ProcessValue <- "bottleTypeSelection"
   Button "Button_1" at 0,414 size 99x66; TextOff 'Start'
      on Press: function_b14e0dd5("keyGrup_a", 0)
      Appearance <- "activeStart"
   Button "Button_2" at 100,414 size 99x66; TextOff 'Stop'
      on Press: function_b14e0dd5("keyGrup_a", 1)
   Button "Button_3" at 200,414 size 99x66; TextOff 'Hardware Param K3'
      on Press: function_b14e0dd5("keyGrup_a", 2)
   Button "Button_4" at 300,414 size 99x66; TextOff 'DW Status K4'
      on Press: function_b14e0dd5("keyGrup_a", 3)
   Button "Button_5" at 400,414 size 99x66; TextOff 'V_EBI Setup K5'
      on Press: function_b14e0dd5("keyGrup_a", 4)
   Button "Button_6" at 500,414 size 200x66; TextOff 'Accept Selection'
      on Press: function_b14e0dd5("bottleAccSelect", 0)
   Button "Button_8" at 701,414 size 99x66; TextOff 'Main'
      on Click: ActivateScreen("107_TRENDS_A", 0)
   TextField "Text field_12" at 204,40 size 166x33; Text 'Speed / 620ml bottle'

screen "116_MESSAGES" 800x480, template "style_1"
   AlarmView "Alarm view_1" at 11,45 size 776x356
   Button "Button_4" at 300,414 size 99x66; TextOff 'DW Status K4'
      on Press: function_b14e0dd5("keyGrup_a", 3)
   Button "Button_5" at 400,414 size 99x66; TextOff 'V_EBI Setup K5'
      on Press: function_b14e0dd5("keyGrup_a", 4)
   Button "Button_6" at 500,414 size 99x66; TextOff 'K6'
      on Press: function_b14e0dd5("keyGrup_a", 5)
   Button "Button_7" at 600,414 size 99x66; TextOff 'Software Param K7'
      on Press: function_b14e0dd5("keyGrup_a", 6)
   Button "Button_8" at 701,414 size 99x66; TextOff 'Main'
      on Click: ActivateScreen("107_TRENDS_A", 0)
   Button "Button_1" at 0,414 size 99x66; TextOff 'Start'
      on Press: function_b14e0dd5("keyGrup_a", 0)
      Appearance <- "activeStart"
   Button "Button_2" at 100,414 size 99x66; TextOff 'Stop'
      on Press: function_b14e0dd5("keyGrup_a", 1)
   Button "Button_3" at 200,414 size 99x66; TextOff 'Stop / K3'
      on Press: function_b14e0dd5("keyGrup_a", 2)

screen "114_PASSWORDS" 800x480, template "style_1"
   Button "Button_4" at 300,414 size 99x66; TextOff 'DW Status K4'
      on Press: function_b14e0dd5("keyGrup_a", 3)
   Button "Button_5" at 400,414 size 99x66; TextOff 'V_EBI Setup K5'
      on Press: function_b14e0dd5("keyGrup_a", 4)
   Button "Button_6" at 500,414 size 99x66; TextOff 'K6'
      on Press: function_b14e0dd5("keyGrup_a", 5)
   Button "Button_7" at 600,414 size 99x66; TextOff 'Software Param K7'
      on Press: function_b14e0dd5("keyGrup_a", 6)
   Button "Button_8" at 701,414 size 99x66; TextOff 'Main'
      on Click: ActivateScreen("107_TRENDS_A", 0)
   UserView "User view_1" at 19,47 size 761x338
   Button "Button_1" at 0,414 size 99x66; TextOff 'Start'
      on Press: function_b14e0dd5("keyGrup_a", 0)
      Appearance <- "activeStart"
   Button "Button_2" at 100,414 size 99x66; TextOff 'Stop'
      on Press: function_b14e0dd5("keyGrup_a", 1)
   Button "Button_3" at 200,414 size 99x66; TextOff 'Stop / K3'
      on Press: function_b14e0dd5("keyGrup_a", 2)

screen "115_TRENDS_B" 800x480, template "style_1"
   TextField "Text field_5" at 175,355 size 469x27; Text 'Parameters and setup only with password !!'
   Button "Button_3" at 200,414 size 99x66; TextOff 'Speed EBI'; Authorization "User administration"
      on Click: ActivateScreen("118_V_EBI_SETUP", 0)
   Button "Button_4" at 300,414 size 99x66; TextOff 'DW Status Inliner'; Authorization "User administration"
      on Click: ActivateScreen("108_INLINER_1", 0)
   Button "Button_5" at 400,414 size 99x66; TextOff 'V_EBI Setup Software Param'; Authorization "User administration"
      on Click: ActivateScreen("119_SOFTWARE_PAR_1", 0)
   Button "Button_6" at 500,414 size 99x66; TextOff 'Hardware Param'; Authorization "User administration"
      on Click: ActivateScreen("105_HARDWARE_PAR_1", 0)
   Button "Button_7" at 600,414 size 99x66; TextOff 'Software Param Passwords'; Authorization "User administration"
      on Click: ActivateScreen("114_PASSWORDS", 0)
   Button "Button_8" at 701,414 size 99x66; TextOff 'Main'
      on Click: ActivateScreen("107_TRENDS_A", 0)
   TextField "Text field_1" at 18,381 size 58x27; Text 'Speed / Filler :'
   TextField "Text field_2" at 594,381 size 58x27; Text 'Speed / EBI :'
   TextField "Text field_3" at 123,379 size 70x27; Text 'Speed / 000 b/h'
   TextField "Text field_4" at 698,379 size 70x27; Text 'Speed / 000 b/h'
   TrendView "Trend view_1" at 9,67 size 785x283
   IOField "I/O field_1" at 74,379 size 47x32; FormatPattern 99999
      ProcessValue <- "speedFiller"
   IOField "I/O field_2" at 651,379 size 47x32; FormatPattern 99999
      ProcessValue <- "speedEBI"
   Button "Button_9" at 6,357 size 786x56; TextOff 'monitor'
      on Click: ActivateScreen("121_DISPLAY_STATUS", 0)
   TextField "Text field_12" at 22,30 size 166x33; Text 'Speed / 620ml bottle'
   Button "Button_1" at 0,414 size 99x66; TextOff 'Start'
      on Press: function_b14e0dd5("keyGrup_a", 0)
      Appearance <- "activeStart"
   Button "Button_2" at 100,414 size 99x66; TextOff 'Stop'
      on Press: function_b14e0dd5("keyGrup_a", 1)

screen "122_DW_STATUS" 800x480, template "style_1"
   TextField "Text field_1" at 56,62 size 288x29; Text 'Speed / Status and modify Datawords'
   Button "Button_8" at 701,414 size 99x66; TextOff 'Main / Back'
      on Click: ActivateScreen("119_SOFTWARE_PAR_1", 0)
   TextField "Text field_2" at 56,129 size 60x27; Text 'Speed / DBnr :'
   TextField "Text field_3" at 271,129 size 66x27; Text 'Speed / DWnr :'
   TextField "Text field_4" at 56,171 size 84x27; Text 'Speed / Decimal :'
   TextField "Text field_5" at 56,211 size 124x27; Text 'Speed / Hexadecimal :'
   TextField "Text field_6" at 56,251 size 70x27; Text 'Speed / Binary :'
   TextField "Text field_7" at 520,126 size 225x195; Text 'Speed Caution !!! Changes may have big consequences only make changes when the function of the dataword is well understood'
   IOField "I/O field_1" at 148,126 size 92x33; FormatPattern 999999
      ProcessValue <- "dbNumber"
   IOField "I/O field_2" at 356,126 size 92x33; FormatPattern 999999
      ProcessValue <- "dwNumber"
   IOField "I/O field_3" at 196,168 size 252x33; FormatPattern 999999
      ProcessValue <- "statusDataWords"
   IOField "I/O field_4" at 196,208 size 252x33; FormatPattern FFFFFFFF
      ProcessValue <- "statusDataWords"
   IOField "I/O field_5" at 139,248 size 309x33; FormatPattern 1111111111111111
      ProcessValue <- "statusDataWords"
   Button "Button_1" at 0,414 size 99x66; TextOff 'Start'
      on Press: function_b14e0dd5("keyGrup_a", 0)
      Appearance <- "activeStart"
   Button "Button_2" at 100,414 size 99x66; TextOff 'Stop'
      on Press: function_b14e0dd5("keyGrup_a", 1)

screen "118_V_EBI_SETUP" 800x480, template "style_1"
   TextField "Text field_1" at 43,29 size 148x50; Text 'Speed Speed regulation EBI'
   Button "Button_4" at 300,414 size 99x66; TextOff 'DW Status'; Authorization "User administration"
      on Click: ActivateScreen("122_DW_STATUS", 0)
   Button "Button_5" at 400,414 size 99x66; TextOff 'V_EBI Setup K5'
      on Press: function_b14e0dd5("keyGrup_a", 4)
   Button "Button_6" at 500,414 size 99x66; TextOff 'Software Param'; Authorization "User administration"
      on Click: ActivateScreen("119_SOFTWARE_PAR_1", 0)
   Button "Button_7" at 600,414 size 99x66; TextOff 'Software Param Inliner page 1'; Authorization "User administration"
      on Click: ActivateScreen("108_INLINER_1", 0)
   Button "Button_8" at 701,414 size 99x66; TextOff 'Main'
      on Click: ActivateScreen("107_TRENDS_A", 0)
   TextField "Text field_2" at 43,91 size 112x27; Text 'Speed / Speed filler :'
   TextField "Text field_3" at 43,122 size 106x27; Text 'Speed / Speed EBI :'
   TextField "Text field_4" at 43,153 size 147x27; Text 'Speed / Lim.over.nomin :'
   TextField "Text field_5" at 43,184 size 161x27; Text 'Speed / Lim.under.nomin :'
   TextField "Text field_6" at 43,215 size 140x27; Text 'Speed / Correction.fact :'
   TextField "Text field_7" at 43,279 size 152x27; Text 'Speed / Max. Speed EBI :'
   TextField "Text field_8" at 43,310 size 148x27; Text 'Speed / Min. Speed EBI :'
   TextField "Text field_9" at 43,371 size 116x27; Text 'Speed / Base Speed :'
   Button "btn_minimSpeed" at 394,104 size 99x73; TextOff 'Stop Minim Speed'
      on Press: function_b14e0dd5("btn_speedchange", 0)
   Button "btn_nominSpeed" at 394,200 size 99x73; TextOff 'Stop Nomin. Speed'
      on Press: function_b14e0dd5("btn_speedchange", 1)
   Button "btn_maximSpeed" at 394,296 size 99x73; TextOff 'Stop Maxim. Speed'
      on Press: function_b14e0dd5("btn_speedchange", 2)
   IOField "I/O field_8" at 575,37 size 73x33; FormatPattern 999999
      ProcessValue <- "speedFiller"
   IOField "I/O field_9" at 672,37 size 73x33; FormatPattern 999999
      ProcessValue <- "speedEBI"
   IOField "I/O field_1" at 246,88 size 73x33; FormatPattern 999999
      ProcessValue <- "speedFiller"
   IOField "I/O field_2" at 246,119 size 73x33; FormatPattern 999999
      ProcessValue <- "speedEBI"
   IOField "I/O field_3" at 246,150 size 73x33; FormatPattern 999999
      ProcessValue <- "limOverNomin"
   IOField "I/O field_4" at 246,181 size 73x33; FormatPattern 999999
      ProcessValue <- "limUnderNomin"
   IOField "I/O field_5" at 246,212 size 73x33; FormatPattern 999999
      ProcessValue <- "correctionFact"
   IOField "I/O field_6" at 246,276 size 73x33; FormatPattern 999999
      ProcessValue <- "maxSpeedEBI"
   IOField "I/O field_7" at 246,307 size 73x33; FormatPattern 999999
      ProcessValue <- "minSpeedEBI"
   IOField "I/O field_10" at 246,368 size 73x33; FormatPattern 999999
      ProcessValue <- "baseSpeed"
   TextField "Text field_12" at 377,37 size 166x33; Text 'Speed / 620ml bottle'
   Bar "filler_speed" at 575,79 size 73x289; MinimumValue 0; MaximumValue 50
      ProcessValue <- "speedFiller"
   TextField "Text field_10" at 583,371 size 58x27; Text 'Speed / Filler'
   TextField "Text field_11" at 672,371 size 58x27; Text 'Speed / EBI'
   Bar "ebi_speed" at 672,79 size 73x289; MinimumValue 0; MaximumValue 50
      ProcessValue <- "speedEBI"
   Button "Button_1" at 0,414 size 99x66; TextOff 'Start'
      on Press: function_b14e0dd5("keyGrup_a", 0)
      Appearance <- "activeStart"
   Button "Button_2" at 100,414 size 99x66; TextOff 'Stop'
      on Press: function_b14e0dd5("keyGrup_a", 1)
   Button "Button_3" at 200,414 size 99x66; TextOff 'Stop / K3'
      on Press: function_b14e0dd5("keyGrup_a", 2)

screen "119_SOFTWARE_PAR_1" 800x480, template "style_1"
   TextField "Text field_1" at 25,36 size 152x27; Text 'Speed / Parameter status'
   Button "Button_4" at 300,414 size 99x66; TextOff 'DW Status'; Authorization "User administration"
      on Click: ActivateScreen("122_DW_STATUS", 0)
   Button "Button_5" at 400,414 size 99x66; TextOff 'V_EBI Setup V_EBI setup'; Authorization "User administration"
      on Click: ActivateScreen("118_V_EBI_SETUP", 0)
   Button "Button_6" at 500,414 size 99x66; TextOff 'Inliner setup'; Authorization "User administration"
      on Click: ActivateScreen("108_INLINER_1", 0)
   Button "Button_7" at 600,414 size 99x66; TextOff 'Software Param Software page 2'; Authorization "User administration"
      on Click: ActivateScreen("123_SOFTWARE_PAR_2", 0)
   Button "Button_8" at 701,414 size 99x66; TextOff 'Main'
      on Click: ActivateScreen("107_TRENDS_A", 0)
   TextField "Text field_2" at 25,79 size 97x27; Text 'Speed / PLC input :'
   TextField "Text field_3" at 25,110 size 107x27; Text 'Speed / PLC calcul. :'
   TextField "Text field_4" at 25,141 size 105x27; Text 'Speed / PLC +fact. :'
   TextField "Text field_5" at 25,172 size 146x27; Text 'Speed / Correction fact. :'
   TextField "Text field_6" at 25,203 size 130x27; Text 'Speed / Minim. speed :'
   TextField "Text field_7" at 25,234 size 134x27; Text 'Speed / Maxim. speed :'
   TextField "Text field_8" at 25,265 size 164x27; Text 'Speed / Corr. LL <> nomi :'
   TextField "Text field_9" at 25,296 size 155x27; Text 'Speed / Corr. L <> nomi :'
   Bar "Bar_1" at 451,84 size 102x289; MinimumValue 0; MaximumValue 1000
      ProcessValue <- "plc_Input"
   Bar "Bar_2" at 553,96 size 33x265; MinimumValue 0; MaximumValue 1000
      ProcessValue <- "plc_Calc"
   IOField "I/O field_8" at 499,33 size 54x33; FormatPattern 999999
      ProcessValue <- "plc_Input"
   IOField "I/O field_9" at 552,33 size 54x33; FormatPattern 999999
      ProcessValue <- "plc_Calc"
   TextField "Text field_10" at 473,372 size 58x27; Text 'Speed / PLC in'
   TextField "Text field_11" at 541,372 size 58x27; Text 'Speed / calc'
   IOField "I/O field_1" at 213,76 size 73x33; FormatPattern 999999
      ProcessValue <- "plc_Input"
   IOField "I/O field_2" at 213,107 size 73x33; FormatPattern 999999
      ProcessValue <- "plc_Calc"
   IOField "I/O field_3" at 213,138 size 73x33; FormatPattern 999999
      ProcessValue <- "plc_+fact"
   IOField "I/O field_4" at 213,169 size 73x33; FormatPattern 999999
      ProcessValue <- "correctionFact"
   IOField "I/O field_5" at 213,200 size 73x33; FormatPattern 999999
      ProcessValue <- "minim_Speed"
   IOField "I/O field_6" at 213,231 size 73x33; FormatPattern 999999
      ProcessValue <- "maxim_Speed"
   IOField "I/O field_7" at 213,262 size 73x33; FormatPattern 999999
      ProcessValue <- "corrLL"
   IOField "I/O field_10" at 213,293 size 73x33; FormatPattern 999999
      ProcessValue <- "corrL"
   IOField "I/O field_11" at 605,33 size 54x33; FormatPattern 999999
      ProcessValue <- "plc_+fact"
   IOField "I/O field_12" at 658,33 size 54x33; FormatPattern 999999
      ProcessValue <- "frequency"
   Bar "Bar_3" at 586,96 size 33x265; MinimumValue 0; MaximumValue 1000
      ProcessValue <- "plc_+fact"
   Bar "Bar_4" at 619,84 size 90x289; MinimumValue 0; MaximumValue 100
      ProcessValue <- "frequency"
   TextField "Text field_12" at 574,372 size 58x27; Text 'Speed / +fact'
   TextField "Text field_13" at 636,372 size 58x27; Text 'Speed / freq'
   TextField "Text field_14" at 25,327 size 159x27; Text 'Speed / Corr. H <> nomi :'
   TextField "Text field_15" at 25,358 size 172x27; Text 'Speed / Corr. HH <> nomi :'
   IOField "I/O field_13" at 213,324 size 73x33; FormatPattern 999999
      ProcessValue <- "corrH"
   IOField "I/O field_14" at 213,355 size 73x33; FormatPattern 999999
      ProcessValue <- "corrHH"
   Button "Button_1" at 0,414 size 99x66; TextOff 'Start'
      on Press: function_b14e0dd5("keyGrup_a", 0)
      Appearance <- "activeStart"
   Button "Button_2" at 100,414 size 99x66; TextOff 'Stop'
      on Press: function_b14e0dd5("keyGrup_a", 1)
   Button "Button_3" at 200,414 size 99x66; TextOff 'Stop / K3'
      on Press: function_b14e0dd5("keyGrup_a", 2)
   SymbolicIOField "Symbolic I/O field_2" at 213,33 size 197x32; TextOn '1'; TextOff '0'; TextList "motor_selection"
      ProcessValue <- "param_select"

screen "123_SOFTWARE_PAR_2" 800x480, template "style_1"
   TextField "Text field_1" at 25,36 size 152x27; Text 'Speed / Parameter status'
   Button "Button_4" at 300,414 size 99x66; TextOff 'DW Status'; Authorization "User administration"
      on Click: ActivateScreen("122_DW_STATUS", 0)
   Button "Button_5" at 400,414 size 99x66; TextOff 'V_EBI Setup V_EBI setup'; Authorization "User administration"
      on Click: ActivateScreen("118_V_EBI_SETUP", 0)
   Button "Button_6" at 500,414 size 99x66; TextOff 'Inliner setup'; Authorization "User administration"
      on Click: ActivateScreen("108_INLINER_1", 0)
   Button "Button_7" at 600,414 size 99x66; TextOff 'Software Param Software page 1'; Authorization "User administration"
      on Click: ActivateScreen("119_SOFTWARE_PAR_1", 0)
   Button "Button_8" at 701,414 size 99x66; TextOff 'Main'
      on Click: ActivateScreen("107_TRENDS_A", 0)
   TextField "Text field_2" at 25,79 size 97x27; Text 'Speed / PLC input :'
   TextField "Text field_3" at 25,110 size 107x27; Text 'Speed / PLC calcul. :'
   TextField "Text field_4" at 25,141 size 105x27; Text 'Speed / PLC +fact. :'
   TextField "Text field_5" at 25,172 size 146x27; Text 'Speed / Correction fact. :'
   TextField "Text field_6" at 25,203 size 131x27; Text 'Speed / Ramp up soft :'
   TextField "Text field_7" at 25,234 size 155x27; Text 'Speed / Ramp down soft :'
   TextField "Text field_8" at 25,265 size 102x27; Text 'Speed / Fill up low :'
   TextField "Text field_9" at 25,296 size 115x27; Text 'Speed / Fill up nomi :'
   IOField "I/O field_1" at 213,76 size 73x33; FormatPattern 999999
      ProcessValue <- "plc_Input"
   IOField "I/O field_2" at 213,107 size 73x33; FormatPattern 999999
      ProcessValue <- "plc_Calc"
   IOField "I/O field_3" at 213,138 size 73x33; FormatPattern 999999
      ProcessValue <- "plc_+fact"
   IOField "I/O field_4" at 213,169 size 73x33; FormatPattern 999999
      ProcessValue <- "correctionFact"
   IOField "I/O field_5" at 213,200 size 73x33; FormatPattern 999999
      ProcessValue <- "rampUpSoft"
   IOField "I/O field_6" at 213,231 size 73x33; FormatPattern 999999
      ProcessValue <- "rampDownSoft"
   IOField "I/O field_7" at 213,262 size 73x33; FormatPattern 999999
      ProcessValue <- "fillUpLow"
   IOField "I/O field_10" at 213,293 size 73x33; FormatPattern 999999
      ProcessValue <- "fillUpNomi"
   SymbolicIOField "param_motorSelection" at 213,33 size 197x32; TextOn '1'; TextOff '0'; TextList "motor_selection"
      ProcessValue <- "param_select"
   TextField "Text field_14" at 25,327 size 111x27; Text 'Speed / Fill up high :'
   TextField "Text field_15" at 25,358 size 113x27; Text 'Speed / Fill up maxi :'
   IOField "I/O field_13" at 213,324 size 73x33; FormatPattern 999999
      ProcessValue <- "fillUpHigh"
   IOField "I/O field_14" at 213,355 size 73x33; FormatPattern 999999
      ProcessValue <- "fillUpMaxi"
   Button "Button_1" at 0,414 size 99x66; TextOff 'Start'
      on Press: function_b14e0dd5("keyGrup_a", 0)
      Appearance <- "activeStart"
   Button "Button_2" at 100,414 size 99x66; TextOff 'Stop'
      on Press: function_b14e0dd5("keyGrup_a", 1)
   Button "Button_3" at 200,414 size 99x66; TextOff 'Stop / K3'
      on Press: function_b14e0dd5("keyGrup_a", 2)
   Bar "Bar_1" at 451,84 size 102x289; MinimumValue 0; MaximumValue 1000
      ProcessValue <- "plc_Input"
   Bar "Bar_2" at 553,96 size 33x265; MinimumValue 0; MaximumValue 1000
      ProcessValue <- "plc_Calc"
   IOField "I/O field_8" at 499,33 size 54x33; FormatPattern 999999
      ProcessValue <- "plc_Input"
   IOField "I/O field_9" at 552,33 size 54x33; FormatPattern 999999
      ProcessValue <- "plc_Calc"
   TextField "Text field_10" at 473,372 size 58x27; Text 'Speed / PLC in'
   TextField "Text field_11" at 541,372 size 58x27; Text 'Speed / calc'
   IOField "I/O field_11" at 605,33 size 54x33; FormatPattern 999999
      ProcessValue <- "plc_+fact"
   IOField "I/O field_12" at 658,33 size 54x33; FormatPattern 999999
      ProcessValue <- "frequency"
   Bar "Bar_3" at 586,96 size 33x265; MinimumValue 0; MaximumValue 1000
      ProcessValue <- "plc_+fact"
   Bar "Bar_4" at 619,84 size 90x289; MinimumValue 0; MaximumValue 100
      ProcessValue <- "frequency"
   TextField "Text field_12" at 574,372 size 58x27; Text 'Speed / +fact'
   TextField "Text field_13" at 636,372 size 58x27; Text 'Speed / freq'

screen "121_DISPLAY_STATUS" 800x480, template "style_1"
   Button "Button_8" at 701,414 size 99x66; TextOff 'Main'
      on Click: ActivateScreen("107_TRENDS_A", 0)
   Circle "Circle_1" at 16,339 size 63x63
      Appearance <- "emc_1"
   TextField "Text field_4" at 40,95 size 74x27; Text 'Speed / Standby'
   TextField "Text field_1" at 40,119 size 79x27; Text 'Speed / Overload'
   TextField "Text field_2" at 40,143 size 76x27; Text 'Speed / Running'
   TextField "Text field_3" at 40,167 size 76x27; Text 'Speed / Warning'
   TextField "Text field_5" at 40,191 size 58x27; Text 'Speed / Fault'
   Button "Button_1" at 0,414 size 99x66; TextOff 'Start'
      on Press: function_b14e0dd5("keyGrup_a", 0)
      Appearance <- "activeStart"
   Button "Button_2" at 100,414 size 99x66; TextOff 'Stop'
      on Press: function_b14e0dd5("keyGrup_a", 1)
   Bar "Bar_1" at 701,50 size 76x340; MinimumValue 0; MaximumValue 42
      ProcessValue <- "speedFiller"
      Appearance <- "speedFiller"
   TextField "Text field_6" at 80,372 size 143x27; Text 'Speed / Emergency Stop'
   Circle "Circle_7" at 230,135 size 29x29
      Appearance <- "state_mot101"
   Circle "Circle_12" at 426,190 size 29x29
      Appearance <- "state_mot106"
   Circle "Circle_13" at 616,29 size 29x29
      Appearance <- "state_mot104"
   Circle "Circle_14" at 483,90 size 29x29
      Appearance <- "state_mot103"
   Circle "Circle_15" at 152,40 size 29x29
      Appearance <- "state_mot102"
   Circle "Circle_16" at 145,265 size 43x43
      Appearance <- "ebi_state"
   Circle "Circle_17" at 482,272 size 53x53
      Appearance <- "filler_state"
   Circle "Circle_30" at 629,141 size 29x29
      Appearance <- "state_mot105"
   Group "Group_1" at 313,257 size 37x34
   Group "Group_3" at 140,177 size 37x34
   Group "Group_2" at 321,94 size 37x34
   Circle "Circle_8" at 332,201 size 29x29
      Appearance <- "state_mot107"
   Group "Group" at 496,326 size 156x80
   Group "Group_4" at 366,325 size 160x69
   Group "Group_5" at 201,38 size 447x74
   Circle "Circle_11" at 324,257 size 15x15
      Appearance <- "emc_3"
   Circle "Circle_23" at 324,276 size 15x15
      Appearance <- "emc_3"
   Circle "Circle_24" at 313,266 size 15x15
      Appearance <- "emc_3"
   Circle "Circle_25" at 335,266 size 15x15
      Appearance <- "emc_3"
   Rectangle "Rectangle_2" at 317,262 size 28x25
      Appearance <- "emc_3"
   Circle "Circle_31" at 151,177 size 15x15
      Appearance <- "emc_4"
   Circle "Circle_32" at 151,196 size 15x15
      Appearance <- "emc_4"
   Circle "Circle_33" at 140,186 size 15x15
      Appearance <- "emc_4"
   Circle "Circle_34" at 162,186 size 15x15
      Appearance <- "emc_4"
   Rectangle "Rectangle_4" at 144,182 size 28x25
      Appearance <- "emc_4"
   Circle "Circle_26" at 332,94 size 15x15
      Appearance <- "emc_2"
   Circle "Circle_27" at 332,113 size 15x15
      Appearance <- "emc_2"
   Circle "Circle_28" at 321,103 size 15x15
      Appearance <- "emc_2"
   Circle "Circle_29" at 343,103 size 15x15
      Appearance <- "emc_2"
   Rectangle "Rectangle_3" at 325,99 size 28x25
      Appearance <- "emc_2"
*)